SUBAPPLICATION HandshakePatternDemo (* Handshake pattern demo: Requester (Plug) coupled to Responder (Socket) via a single EVENT_HS adapter connection *)
  (* Standard: 61499-2; Description: Copyright (c) 2026 Meisterschulen am Ostbahnhof This program and the accompanying materials are made available under the terms of the Eclipse Public License 2.0 which is available at https://www.eclipse.org/legal/epl-2.0/ SPDX-License-Identifier: EPL-2.0 *)
  (* Version 1.0, 2026-08-31, Franz Höpfinger, Meisterschulen am Ostbahnhof, Handshake design pattern (IEC 61499 primer course, Module 6, Valeriy Vyatkin), demo application *)
  PACKAGE Meins::DesingPatterns::HandshakePattern;
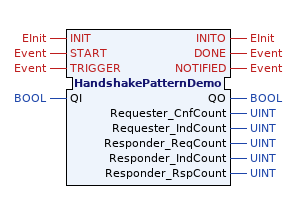
  EVENT_INPUT
    INIT : EInit; (* Initialization Request *)
    START; (* Trigger the Requester to send a REQ *)
    TRIGGER; (* Trigger the Responder to send an unsolicited IND *)
  END_EVENT
  EVENT_OUTPUT
    INITO : EInit; (* Initialization Confirm *)
    DONE; (* Requester received the CNF for the last REQ *)
    NOTIFIED; (* Requester received an IND and answered with RSP *)
  END_EVENT
  VAR_INPUT
    QI : BOOL; (* Input event qualifier *)
  END_VAR
  VAR_OUTPUT
    QO : BOOL; (* Output event qualifier *)
    Requester_CnfCount : UINT; (* Requester: number of CNF received *)
    Requester_IndCount : UINT; (* Requester: number of IND received / RSP sent *)
    Responder_ReqCount : UINT; (* Responder: number of REQ received *)
    Responder_IndCount : UINT; (* Responder: number of IND sent *)
    Responder_RspCount : UINT; (* Responder: number of RSP received *)
  END_VAR
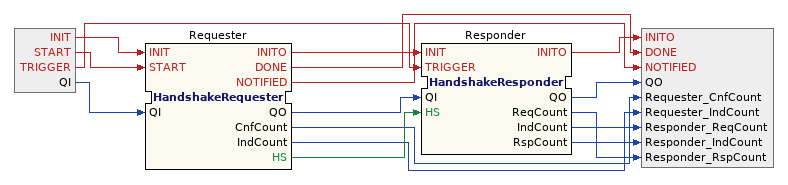
  FBS
    Requester : Meins::DesingPatterns::HandshakePattern::HandshakeRequester;
    Responder : Meins::DesingPatterns::HandshakePattern::HandshakeResponder;
  END_FBS
  EVENT_CONNECTIONS
    START TO Requester.START;
    TRIGGER TO Responder.TRIGGER;
    Requester.DONE TO DONE;
    Requester.NOTIFIED TO NOTIFIED;
    INIT TO Requester.INIT;
    Requester.INITO TO Responder.INIT;
    Responder.INITO TO INITO;
  END_CONNECTIONS
  DATA_CONNECTIONS
    QI TO Requester.QI;
    Requester.QO TO Responder.QI;
    Responder.QO TO QO;
    Requester.CnfCount TO Requester_CnfCount;
    Requester.IndCount TO Requester_IndCount;
    Responder.ReqCount TO Responder_ReqCount;
    Responder.IndCount TO Responder_IndCount;
    Responder.RspCount TO Responder_RspCount;
  END_CONNECTIONS
  ADAPTER_CONNECTIONS
    Requester.HS TO Responder.HS; (* The single Handshake adapter connection replacing REQ/CNF/IND/RSP as four separate event links (Requester=Plug is the Source, Responder=Socket is the Destination) *)
  END_CONNECTIONS
END_SUBAPPLICATION
